TYPE HmiFeedback :
STRUCT
	Control		: RemoteControl;
	Feedback	: RemoteFeedback;
END_STRUCT
END_TYPE

(* stored: Version 1.1.0.1, ProductVersion 3.1.4020.12
   DUT HmiFeedback: Id {d464d86d-062f-4988-a6e1-4ba556c79c34} *)
